# B&R Automation Studio project mappViewSample
Automation Studio 4.5.4.123 SP; technology packages: mapp 5.8.0, mappView 5.8.0

## Configuration Config1

CPU PC_any, AutomationRuntime C4.90, Build 4.1.2, Safety 0.0, Vc V4.72.2

### Task classes (Cpu.sw)
```
Cyclic#1 (cycle 10000 us):
  Program <- Program.prg
Binaries: TCLang, udbdef, mvLoader, arsvcreg, TCData, sysconf, ashwd, ashwac, asfw, iomap, Config, Role, TC, Report, arconfig, User, OpcUaMap
Libraries: MpReport, MpBase, MpWebXs, AsArSdm, runtime, sys_lib, astime, asieccon, fileio
```

### Hardware
```
PC : PC_any v1.1.0.0 (OrderNumber=PC)
  ConfigurationID = mappViewSample_Config1
  Cyclic1Duration = 10000
  FileDevice1
  FileDeviceName1 = SIM_DEVICE
  FileDevicePath1 = C:\Temp
  ActivateOpcUa = 1
  OpcUaInformationModels_PV_Version = 1
```

### Config.mpaudittrail - PC/mappServices/Config.mpaudittrail
```
Element gAuditTrail (Type=mpaudittrail)
  Audit:
    Events:
      [0] = 16
      [1] = 2
      [2] = 18
      [3] = 19
    TextSource = TXT
      OutputFormat = MpAudit/Event/Root
  Monitor:
    0:
      pv = ::TestVar1
      id = 
```

### Config.mpwebxs - PC/mappServices/Config.mpwebxs
```
Element WebXs (Type=mpwebxs)
```

### Report.mpreportcore - PC/mappServices/Report.mpreportcore
```
Element gReport (Type=mpreportcore)
  MpReport:
    Settings:
      ResourceDeviceName = SIM_DEVICE
      LanguageDependent:
        [0]:
          Language = en
    PageLayouts:
      [0]:
        Name = Default
        Margins = 3
    Styles:
      Text:
        [0]:
          Name = Default
        [1]:
          Name = Orange_20
          Size = 20
          Color = FF9900
        [2]:
          Name = Bold_11
          Style = 1
          Size = 11
      Table:
        [0]:
          Name = Default
        [1]:
          Name = Weight_0
          BorderWidth = 0
      Line:
        [0]:
          Name = Default
      Chart:
        PieChart:
          [0]:
            Name = Default
        LineChart:
          [0]:
            Name = Default
        BarChart:
          [0]:
            Name = Default
    Tables:
      [0]:
        Name = ProdutctionTab
        TableStyle = Default
        TextStyle = Default
        [0]:
          [0] = TextId
            Source = Nr.
            Width = 10
          [1] = TextId
            Source = Product Name
            Width = 30
          [2] = TextId
            Source = Batch Size
            Width = 20
          [3] = TextId
            Source = Quality rate
            Width = 20
          [4] = TextId
            Source = Time
            Width = 20
        [1]:
          [0] = TextId
            Source = 1
            Width = 10
          [1] = TextId
            Source = Product Yellow
            Width = 30
          [2] = ValueId
            Value:
              ProcessVariable = ::TestVar1
            Width = 20
          [3] = ValueId
            Value:
              ProcessVariable = ::TestVar2
            Width = 20
          [4] = ValueId
            Value:
              ProcessVariable = ::TestVar3
            Width = 20
        [2]:
          [0] = TextId
            Source = 1
            Width = 10
          [1] = TextId
            Source = Product Yellow
            Width = 30
          [2] = ValueId
            Value:
              ProcessVariable = ::TestVar1
            Width = 20
          [3] = ValueId
            Value:
              ProcessVariable = ::TestVar2
            Width = 20
          [4] = ValueId
            Value:
              ProcessVariable = ::TestVar3
            Width = 20
        [3]:
          [0] = TextId
            Source = 1
            Width = 10
          [1] = TextId
            Source = Product Yellow
            Width = 30
          [2] = ValueId
            Value:
              ProcessVariable = ::TestVar1
            Width = 20
          [3] = ValueId
            Value:
              ProcessVariable = ::TestVar2
            Width = 20
          [4] = ValueId
            Value:
              ProcessVariable = ::TestVar3
            Width = 20
        [4]:
          [0] = TextId
            Source = 1
            Width = 10
          [1] = TextId
            Source = Product Yellow
            Width = 30
          [2] = ValueId
            Value:
              ProcessVariable = ::TestVar1
            Width = 20
          [3] = ValueId
            Value:
              ProcessVariable = ::TestVar2
            Width = 20
          [4] = ValueId
            Value:
              ProcessVariable = ::TestVar3
            Width = 20
      [1]:
        Name = CompanyTab
        TableStyle = Weight_0
        TextStyle = Default
        [0]:
          [0] = TextId
            Source = Company Name
            Width = 50
            TextStyleReference = LocalTextStyle
              TextStyle = Bold_11
          [1] = TextId
            Source = ABC
            Width = 50
        [1]:
          [0] = TextId
            Source = Date
            Width = 50
            TextStyleReference = LocalTextStyle
              TextStyle = Bold_11
        [2]:
          [0] = TextId
            Source = Shift
            Width = 50
            TextStyleReference = LocalTextStyle
              TextStyle = Bold_11
          [1] = TextId
            Source = 7am-3pm
            Width = 50
        [3]:
          [0] = TextId
            Source = Operator
            Width = 50
            TextStyleReference = LocalTextStyle
              TextStyle = Bold_11
          [1] = TextId
            Source = John Doe
            Width = 50
    Charts:
      [0] = LineChart
        Name = ChartLine
        Heading = SingleText
          Text = Line Chart
          HorizontalAlign = 1
          TextStyle = Bold_11
        ChartStyle = Default
        TextStyle = Bold_11
        ShowLegend = 2
        Y[0]:
          Name = Temperatur
          Label = Temperatur
          NumberOfGridLines = 4
        XAxis:
          ProcessVariable = ::ChartXaxis
        [0]:
          YAxis = Temperatur
          Value:
            ProcessVariable = ::ChartData
          LegendText = Temperature
      [1]:
        Name = ChartPie
        Heading = SingleText
          Text = Pie Chart
          HorizontalAlign = 1
          TextStyle = Bold_11
        ChartStyle = Default
        TextStyle = Default
        ShowLegend = 2
        [0]:
          Value:
            ProcessVariable = ::TestVar1
          ItemBackColor = FF0000
          LegendText = Red Cake
        [1]:
          Value:
            ProcessVariable = ::TestVar2
          LegendText = Black Cake
    Contents:
      [0]:
        Name = Heading
        [0]:
          Text = Daily Production Report
          HorizontalAlign = 1
          TextStyle = Orange_20
      [1]:
        Name = Line
        [0] = Line
          LineStyle = Default
      [2]:
        Name = ProductionTable
        [0] = Table
          Table = ProdutctionTab
      [3]:
        Name = CompanyTable
        [0] = Table
          Table = CompanyTab
      [4]:
        Name = Chart Content
        [0] = Chart
          Chart = ChartPie
          Width = 25
        [1] = Line
          LineStyle = Default
        [2] = Chart
          Chart = ChartLine
          Width = 80
      [5]:
        Name = BuR Image
        [0] = Image
          Image = BuR.jpg
    Reports:
      [0]:
        Name = MyReport
        PageLayout = Default
        Header = Heading
        [0]:
          [0]:
            Content = BuR Image
        [1]:
          Heading:
            Text = 
            HorizontalAlign = 1
            TextStyle = Default
          [0]:
            Content = Line
        [2]:
          [0]:
            Content = CompanyTable
        [3]:
          Heading:
            Text = 
            HorizontalAlign = 1
            TextStyle = Default
          [0]:
            Content = Line
        [4]:
          [0]:
            Content = ProductionTable
        [5]:
          StartOnNewPage = TRUE
          Heading:
            TextStyle = Bold_11
          [0]:
            Content = Chart Content
```

## Logical view

Binary libraries used (declarations not repeated): operator, runtime, astime, AsIecCon, AsArSdm, MpWebXs 5.08.0, MpBase 5.08.0, MpReport 5.08.0, MpAudit 5.07.1

### Global.typ - Global data types
```iecst
TYPE
	typMotor : 	STRUCT
		Position : REAL;
		Acceleration : UINT;
		Velocity : UINT;
		IsVisible : BOOL;
	END_STRUCT;
	ClientInfoType : 	STRUCT
		userId : WSTRING[80];
		isValid : BOOL;
		ipAddress : WSTRING[15];
		languageId : WSTRING[2];
		screenResolution : WSTRING[32];
		slotId : SINT;
	END_STRUCT;
END_TYPE
```

### Global.var - Global variables
```iecst
VAR
	TestVar1 : UINT;
	TestVar2 : INT;
	TestVar3 : REAL;
	ChartData : ARRAY[0..99] OF DINT;
	ChartXaxis : ARRAY[0..99] OF TIME;
END_VAR
```


### Program Logical/Program (IEC)

#### Main.st - Init, cyclic, exit code
```iecst
PROGRAM _INIT
	TestVar1 := 30;

END_PROGRAM

PROGRAM _CYCLIC
	TestVar2 := 100 - TestVar1;
	TestVar3 := TestVar3 + 0.1;

	// Create chart sample data
	ChartData[idx] := idy;
	idy := idy + 1;
	IF(idy > 50) THEN
		idy := 0;
	END_IF
	idx := idx + 1;
	IF(idx > 99) THEN
		idx := 0;
	END_IF
	ChartXaxis[idx] := USINT_TO_TIME(idx);

	MpReportCore_0(MpLink := ADR(gReport), Enable := 1, Name := ADR('MyReport'), Language := ADR('en'), DeviceName := ADR('SIM_DEVICE'));

END_PROGRAM

PROGRAM _EXIT
	 MpReportCore_0(MpLink := ADR(gReport), Enable := 0);
END_PROGRAM
```

#### Variables.var - Local variables
```iecst
VAR
	idy : USINT;
	idx : USINT;
	MpReportCore_0 : MpReportCore;
END_VAR
```

- Visualisation Logical/mappView (not shown)

- Project.language (not shown)

Listed in the project but not available here: Logical/Program/Types.typ
